INTERFACE ISum

(*This method adds two DINT numbers and returns the result in Sum*)
METHOD Sum : DINT;
VAR_INPUT
	Dint1 : DINT;
	Dint2 : DINT;
END_VAR
END_METHOD

END_INTERFACE

(* stored: Version 1.1.0.1, ProductVersion 3.1.4024.6
   Itf ISum: Id {e39d6e09-a369-4129-9752-3448bbb020db}
   Method Sum: Id {2d4a4a07-7b2b-47df-8e72-927c70ac455b} *)
